FUNCTION_BLOCK EM_LogicExample_1 EXTENDS FB_EM_Base IMPLEMENTS ITF_EM_LogicExample1
VAR_INPUT	
	i_stMachineCommands				: ST_UN_Machine100_Cmd;
END_VAR
VAR
// Variables
	s_bStaStateOfSomething			: BOOL;
	s_bStaStateOfSomething2			: BOOL;
	s_bStaStateOfSomething3			: BOOL;
	s_bStaStateOfSomething4			: BOOL;
	s_bStaStateOfSomething5			: BOOL;
	s_bStaStateOfSomething6			: BOOL;
	s_bStaStateOfSomething7			: BOOL;
	s_fStaValue						: LREAL;
	s_fStaValueResult				: LREAL;
	
// Config Struct
	s_stConfig						: ST_EM_LogicExample1_Config;
	
// Control modules
	s_cmVirtualMaster				: CM_Servo_Virtual;
	s_cmAxis1						: CM_Servo_Virtual;
	s_cmAxis1Cam					: CM_Servo_CammingAddon(s_cmAxis1);
	s_cmAxis1Fly					: CM_Servo_FlyingSawAddon(s_cmAxis1);
	s_cmWaterInlet					: CM_Valve;
	s_cmBelt						: CM_MotorDol;
	s_cmHeightAdjuster				: CM_MotorDol_AF;
	s_cmVentilator					: CM_MotorVFD_Lenze_i5xx;
	
// Inputs
	s_fbDiSensorPos1				: FB_DigitalInput;
	
// Outputs
	s_fbDoMachineX_Start			: FB_DigitalOutput;
	s_fbAoMachineX_Speed			: FB_AnalogOutput;
	s_fbRedLight					: FB_Light;
	s_fbBlueButton					: FB_PushButtonLight;
	s_fbStackLight					: FB_StackLights;
	
// Alarms
	s_AlmFailure1					: FB_AlarmHandler;
	s_AlmFailure2					: FB_AlarmHandler;
	
// Statistics
	s_fbRunTime_Belt				: FB_RunningTime;
	
END_VAR
VAR CONSTANT
	nCamTableIdAxis1			: UINT := 1;
END_VAR

SUPER^();

METHOD PROTECTED _m_Aborting
VAR_INPUT
	i_rstPML_Status			: REFERENCE TO ST_PackML_Status;
END_VAR
VAR_INST
	
	s_bStaStateComplete1		: BOOL;
END_VAR
i_rstPML_Status.bStateComplete := _m_StopServos(i_bReqStart := i_rstPML_Status.bStateEntry);
END_METHOD

METHOD PROTECTED _m_Alarms
VAR_INST
	s_tonAlmFailure2_DelayedAutoReset	: TON;
END_VAR
SUPER^._m_Alarms();

// Failure 1
s_stConfig.stAlmFailure1.nIDnr		:= 1;
s_stConfig.stAlmFailure1.eAction	:= E_Alarm_Actions.Abort;
s_stConfig.stAlmFailure1.tmDelay	:= T#1S;
s_stConfig.stAlmFailure1.bEnable	:= q_bStaEnabled;
s_AlmFailure1(
	i_bCmdSet	:= s_fbDiSensorPos1.q_bStaInput 
				AND s_bStaStateOfSomething,
	i_sMsgVar1	:= 'Fault code: ',
	//i_sMsgVar2	:= TO_STRING(s_nFaultCode),
	i_rstConfig	:= s_stConfig.stAlmFailure1,
	i_itfAlarmCollector := s_fbAlarmCollector);

	
// Failure 2
s_stConfig.stAlmFailure2.nIDnr	:= 2;
s_stConfig.stAlmFailure2.eAction := E_Alarm_Actions.Suspend;

// Automatic reset timer
s_tonAlmFailure2_DelayedAutoReset(IN := s_AlmFailure2.p_bStaActive AND NOT s_AlmFailure2.p_bStaCmdSet, PT := T#5S);
// Reset the alarm after the delay time
IF s_tonAlmFailure2_DelayedAutoReset.Q THEN
	s_AlmFailure2.m_CmdReset();
END_IF

s_AlmFailure2(
	i_rstConfig	:= s_stConfig.stAlmFailure2,
	i_itfAlarmCollector := s_fbAlarmCollector);
END_METHOD

METHOD PROTECTED _m_Execute
VAR_INPUT
	i_rstPML_Status			: REFERENCE TO ST_PackML_Status;
END_VAR
VAR_INST
	s_eActMode				: E_PackML_Mode;
END_VAR
// Execute only when in a specific mode
s_eActMode := i_rstPML_Status.eActMode;
CASE s_eActMode OF
	E_PackML_Mode.Production: 
		// Execute only when in PRODUCTION mode
		i_rstPML_Status.bStateComplete := _m_Execute_Production(i_bReqStart := i_rstPML_Status.bStateEntry);
				
ELSE
	// Execute in all other modes	
	i_rstPML_Status.bStateComplete := TRUE;
END_CASE
END_METHOD

METHOD PROTECTED _m_Execute_Production : BOOL
VAR_INPUT
	i_bReqStart				: BOOL;
END_VAR
VAR_INST
	s_fbSeqControl			: FB_SeqControl;
	s_eSeqAutoExecute		: E_EM_LogicExample1_Seq_ExecuteProduction;
	s_stSyncMode			: ST_SyncMode;			// Synchronisation mode
	
	
	s_fCalculatedSpeed		: LREAL;		// Calculated VM speed, based on machine setting
	s_fShortestPosition		: LREAL;		
END_VAR
// Sequence exceptions
// n.a.


// Sequencer control
s_fbSeqControl(
	i_bReqStart		:= i_bReqStart, 
	i_rnActSeqStep	:= s_eSeqAutoExecute,
	i_sActSeqStep	:= TO_STRING(s_eSeqAutoExecute));
	
// Sequence	
CASE s_eSeqAutoExecute OF
	
	E_EM_LogicExample1_Seq_ExecuteProduction.Idle:
		;
			
	E_EM_LogicExample1_Seq_ExecuteProduction.Start:
		s_fCalculatedSpeed	:= (360.0 * 1000.0) / 123.4; // 360 degree = 1 product. 
		IF s_cmVirtualMaster.m_StartFF(
			i_bCmdReset		:= s_fbSeqControl.q_bStaEntry, 
			i_fAcceleration	:= s_cmVirtualMaster.q_stParameterSet.fAccelerationMax, 
			i_fDeceleration	:= s_cmVirtualMaster.q_stParameterSet.fDecelerationMax, 
			i_fJerk			:= s_cmVirtualMaster.q_stParameterSet.fJerk, 
			i_fSpeed		:= s_cmVirtualMaster.q_stParameterSet.fVeloFastManual,
			i_sLogHint		:= '',
			i_eBufferMode	:= MC_BufferMode.MC_Aborting) 
		THEN
			s_fbSeqControl.m_ReqStep(E_EM_LogicExample1_Seq_ExecuteProduction.StartWait);
		END_IF
		

	//Wait for 5 seconds
	E_EM_LogicExample1_Seq_ExecuteProduction.StartWait:
		IF s_fbSeqControl.q_tmStepTime> T#5S THEN
			s_fbSeqControl.m_ReqStep(E_EM_LogicExample1_Seq_ExecuteProduction.Step1);
		END_IF

		
	//gear out Slave axis 1 without stopping the axis
	E_EM_LogicExample1_Seq_ExecuteProduction.Step1:
		IF s_cmAxis1.m_GearOut(i_bCmdReset:=s_fbSeqControl.q_bStaEntry) THEN
			s_fbSeqControl.m_ReqStep(E_EM_LogicExample1_Seq_ExecuteProduction.Step1Wait);
		END_IF

		
	//Wait for 5 seconds
	E_EM_LogicExample1_Seq_ExecuteProduction.Step1Wait:
		IF s_fbSeqControl.q_tmStepTime> T#5S THEN
			s_fbSeqControl.m_ReqStep(E_EM_LogicExample1_Seq_ExecuteProduction.Step2);
		END_IF
		
		
	//gear in Slave axis 1 at position
	E_EM_LogicExample1_Seq_ExecuteProduction.Step2:
		IF s_fbSeqControl.q_bStaEntry THEN
			//Enable disable checks. An enabled check gives an NC error when the check condition is true.	
			s_stSyncMode.GearInSyncMode 						:= E_GearInSyncMode.GEARINSYNCMODE_POSITIONBASED;
			s_stSyncMode.GearInSync_CheckMask_MinPos 			:= FALSE;
			s_stSyncMode.GearInSync_CheckMask_MaxPos 			:= FALSE;
			s_stSyncMode.GearInSync_CheckMask_MaxVelo 			:= FALSE;
			s_stSyncMode.GearInSync_CheckMask_MaxAcc 			:= FALSE;
			s_stSyncMode.GearInSync_CheckMask_MaxDec 			:= FALSE;
			s_stSyncMode.GearInSync_CheckMask_MaxJerk 			:= FALSE;
			s_stSyncMode.GearInSync_CheckMask_OvershootPos 		:= FALSE;
			s_stSyncMode.GearInSync_CheckMask_UndershootPos 	:= FALSE;
			s_stSyncMode.GearInSync_CheckMask_OvershootVelo 	:= FALSE;
			s_stSyncMode.GearInSync_CheckMask_UndershootVelo 	:= FALSE;
			s_stSyncMode.GearInSync_CheckMask_OvershootVeloZero := FALSE;
			s_stSyncMode.GearInSync_CheckMask_UndershootVeloZero:= FALSE;
			
			//Optimalization methodes
			s_stSyncMode.GearInSync_OpMask_RollbackLock 		:= TRUE;
			s_stSyncMode.GearInSync_OpMask_InstantStopOnRollback:= TRUE;
			s_stSyncMode.GearInSync_OpMask_PreferConstVelo 		:= TRUE;
			s_stSyncMode.GearInSync_OpMask_IgnoreMasterAcc 		:= TRUE;
		END_IF

		IF s_cmAxis1Fly.m_GearInPos(
			i_bCmdReset				:= s_fbSeqControl.q_bStaEntry, 
			i_fAcceleration			:= s_cmAxis1.q_stParameterSet.fAccelerationMax, 
			i_fDeceleration			:= s_cmAxis1.q_stParameterSet.fDecelerationMax, 
			i_fJerk					:= s_cmAxis1.q_stParameterSet.fJerk, 
			i_fSpeed				:= s_cmAxis1.q_stParameterSet.fVeloMaximum, 
			i_fMasterSyncPosition	:= s_cmVirtualMaster.q_fActualPos + 1000.0, 
			i_fSlaveSyncPosition	:= s_cmAxis1.q_fActualPos + 2000.0, 
			i_stSyncMode			:= s_stSyncMode, 
			i_fSlaveScale			:= 1.0, 
			i_fMasterScale			:= 1.0, 
			i_itfMaster				:= s_cmVirtualMaster) 
		THEN
			s_fbSeqControl.m_ReqStep(E_EM_LogicExample1_Seq_ExecuteProduction.Step2Wait);
		END_IF

		
	//Wait till synchronized
	E_EM_LogicExample1_Seq_ExecuteProduction.Step2Wait:
		IF s_cmAxis1.q_bStaInSync THEN
			s_fbSeqControl.m_ReqStep(E_EM_LogicExample1_Seq_ExecuteProduction.Step3);
		END_IF
		
		
	//gear out Slave axis 1 without stopping the axis when the axis is synchronized
	E_EM_LogicExample1_Seq_ExecuteProduction.Step3:
		IF s_cmAxis1.m_GearOut(i_bCmdReset:=s_fbSeqControl.q_bStaEntry) THEN
			s_fbSeqControl.m_ReqStep(E_EM_LogicExample1_Seq_ExecuteProduction.Step3Wait);
		END_IF

		
	//Wait for 5 seconds
	E_EM_LogicExample1_Seq_ExecuteProduction.Step3Wait:
		IF s_fbSeqControl.q_tmStepTime> T#5S THEN
			s_fbSeqControl.m_ReqStep(E_EM_LogicExample1_Seq_ExecuteProduction.Step4);
		END_IF
		
		
	//gear in Slave axis 1 at speed
	E_EM_LogicExample1_Seq_ExecuteProduction.Step4:
		IF s_fbSeqControl.q_bStaEntry THEN
			//Enable disable checks. An enabled check gives an NC error when the check condition is true.	
			s_stSyncMode.GearInSyncMode 						:= E_GearInSyncMode.GEARINSYNCMODE_POSITIONBASED;
			s_stSyncMode.GearInSync_CheckMask_MinPos 			:= FALSE;
			s_stSyncMode.GearInSync_CheckMask_MaxPos 			:= FALSE;
			s_stSyncMode.GearInSync_CheckMask_MaxVelo 			:= FALSE;
			s_stSyncMode.GearInSync_CheckMask_MaxAcc 			:= FALSE;
			s_stSyncMode.GearInSync_CheckMask_MaxDec 			:= FALSE;
			s_stSyncMode.GearInSync_CheckMask_MaxJerk 			:= FALSE;
			s_stSyncMode.GearInSync_CheckMask_OvershootPos 		:= FALSE;
			s_stSyncMode.GearInSync_CheckMask_UndershootPos 	:= FALSE;
			s_stSyncMode.GearInSync_CheckMask_OvershootVelo 	:= FALSE;
			s_stSyncMode.GearInSync_CheckMask_UndershootVelo 	:= FALSE;
			s_stSyncMode.GearInSync_CheckMask_OvershootVeloZero := FALSE;
			s_stSyncMode.GearInSync_CheckMask_UndershootVeloZero:= FALSE;
			
			//Optimalization methodes
			s_stSyncMode.GearInSync_OpMask_RollbackLock 		:= TRUE;
			s_stSyncMode.GearInSync_OpMask_InstantStopOnRollback:= TRUE;
			s_stSyncMode.GearInSync_OpMask_PreferConstVelo 		:= TRUE;
			s_stSyncMode.GearInSync_OpMask_IgnoreMasterAcc 		:= TRUE;
		END_IF
	
		IF s_cmAxis1Fly.m_GearInSpeed(
			i_bCmdReset		:= s_fbSeqControl.q_bStaEntry, 
			i_fSlaveScale	:= 2.0, 
			i_fMasterScale	:= 1.0, 
			i_stSyncMode	:= s_stSyncMode, 
			i_fAcceleration	:= s_cmAxis1.q_stParameterSet.fAccelerationMax, 
			i_fDeceleration	:= s_cmAxis1.q_stParameterSet.fDecelerationMax, 
			i_fJerk			:= s_cmAxis1.q_stParameterSet.fJerk, 
			i_fSpeed		:= s_cmAxis1.q_stParameterSet.fVeloMaximum, 
			i_itfMaster		:= s_cmVirtualMaster ) 
		THEN
			s_fbSeqControl.m_ReqStep(E_EM_LogicExample1_Seq_ExecuteProduction.Step4Wait);
		END_IF

		
	//Wait till synchronized
	E_EM_LogicExample1_Seq_ExecuteProduction.Step4Wait:
		IF s_cmAxis1.q_bStaInSync THEN
			s_fbSeqControl.m_ReqStep(E_EM_LogicExample1_Seq_ExecuteProduction.Step5);
		END_IF
		
		
	//halt Master and Slave axis => axis will gearout and stopping 
	E_EM_LogicExample1_Seq_ExecuteProduction.Step5:
			IF s_cmVirtualMaster.m_Halt(
				i_bCmdReset		:= s_fbSeqControl.q_bStaEntry,
				i_fDeceleration	:= s_cmVirtualMaster.q_stParameterSet.fDecelerationMax,
				i_fJerk			:= s_cmVirtualMaster.q_stParameterSet.fJerk,
				i_eBufferMode	:= MC_BufferMode.MC_Aborting) 
			AND
				s_cmAxis1.m_Halt(
				i_bCmdReset		:= s_fbSeqControl.q_bStaEntry,
				i_fDeceleration	:= s_cmAxis1.q_stParameterSet.fDecelerationMax,
				i_fJerk			:= s_cmAxis1.q_stParameterSet.fJerk, 
				i_eBufferMode	:= MC_BufferMode.MC_Aborting) 
			THEN
			s_fbSeqControl.m_ReqStep(E_EM_LogicExample1_Seq_ExecuteProduction.Step5Wait);
			END_IF

			
	//Wait till axis standstill
	E_EM_LogicExample1_Seq_ExecuteProduction.Step5Wait:
		IF s_cmAxis1.q_stAxisState.StandStill AND s_cmVirtualMaster.q_stAxisState.StandStill THEN
			s_fbSeqControl.m_ReqStep(E_EM_LogicExample1_Seq_ExecuteProduction.Step6);
		END_IF
			
		
	//Gear in dynamic 
	E_EM_LogicExample1_Seq_ExecuteProduction.Step6:
		IF s_cmAxis1.m_GearInDyn(
			i_bCmdReset		:= s_fbSeqControl.q_bStaEntry, 
			i_fAcceleration	:= s_cmAxis1.q_stParameterSet.fAccelerationMax, 
			i_fDeceleration	:= s_cmAxis1.q_stParameterSet.fDecelerationMax, 
			i_fJerk			:= s_cmAxis1.q_stParameterSet.fJerk, 
			i_fGearRatio	:= 1.0, 
			i_itfMaster		:= s_cmVirtualMaster) 
		THEN
			//No wait step nessary m_GearInDyn give TRUE when axis is coupled
			s_fbSeqControl.m_ReqStep(E_EM_LogicExample1_Seq_ExecuteProduction.Step7);
		END_IF
		
	//Move master relative 
	E_EM_LogicExample1_Seq_ExecuteProduction.Step7:
		IF s_cmVirtualMaster.m_StartRelative(
			i_bCmdReset		:= s_fbSeqControl.q_bStaEntry, 
			i_fAcceleration	:= s_cmVirtualMaster.q_stParameterSet.fAccelerationMax, 
			i_fDeceleration	:= s_cmVirtualMaster.q_stParameterSet.fDecelerationMax, 
			i_fJerk			:= s_cmVirtualMaster.q_stParameterSet.fJerk, 
			i_fSpeed		:= s_cmVirtualMaster.q_stParameterSet.fVeloFastManual, 
			i_fPosition		:= 1000.0,
			i_sLogHint		:= '',
			i_eBufferMode	:= MC_BufferMode.MC_Aborting) 
		THEN
			s_fbSeqControl.m_ReqStep(E_EM_LogicExample1_Seq_ExecuteProduction.Step7Wait);
		END_IF

		
	//Wait for 5 seconds
	E_EM_LogicExample1_Seq_ExecuteProduction.Step7Wait:
		IF s_fbSeqControl.q_tmStepTime> T#5S THEN
			s_fbSeqControl.m_ReqStep(E_EM_LogicExample1_Seq_ExecuteProduction.Step8);
		END_IF
		
		
	//Change gearfactor 
	E_EM_LogicExample1_Seq_ExecuteProduction.Step8:
		IF s_cmAxis1.m_GearInDynGearRatio(i_fGearRatio:= 0.5) THEN
			s_fbSeqControl.m_ReqStep(E_EM_LogicExample1_Seq_ExecuteProduction.Step8Wait);
		END_IF

		
	//Wait for 5 seconds
	E_EM_LogicExample1_Seq_ExecuteProduction.Step8Wait:
		IF s_fbSeqControl.q_tmStepTime> T#5S THEN
			s_fbSeqControl.m_ReqStep(E_EM_LogicExample1_Seq_ExecuteProduction.Step9);
		END_IF
		
		
	//stop Master and Slave axis => axis will gearout and stopping 
	E_EM_LogicExample1_Seq_ExecuteProduction.Step9:
		IF s_cmVirtualMaster.m_Stop(
			i_bCmdReset		:= s_fbSeqControl.q_bStaEntry,
			i_fDeceleration	:= s_cmVirtualMaster.q_stParameterSet.fDecelerationMax,
			i_fJerk			:= s_cmVirtualMaster.q_stParameterSet.fJerk) 
		AND
			s_cmAxis1.m_Stop(
			i_bCmdReset		:= s_fbSeqControl.q_bStaEntry,
			i_fDeceleration	:= s_cmAxis1.q_stParameterSet.fDecelerationMax,
			i_fJerk			:= s_cmAxis1.q_stParameterSet.fJerk) 
		THEN
			s_fbSeqControl.m_ReqStep(E_EM_LogicExample1_Seq_ExecuteProduction.Step10Wait);
		END_IF

		
	//Wait till axis standstill
	E_EM_LogicExample1_Seq_ExecuteProduction.Step10Wait:
		IF s_cmAxis1.q_stAxisState.StandStill AND s_cmVirtualMaster.q_stAxisState.StandStill THEN
			s_fbSeqControl.m_ReqStep(E_EM_LogicExample1_Seq_ExecuteProduction.Step11);
		END_IF
		
		
	//Gear in static 
	E_EM_LogicExample1_Seq_ExecuteProduction.Step11:
		IF s_cmAxis1.m_GearInStatic(
			i_bCmdReset		:= s_fbSeqControl.q_bStaEntry, 
			i_fAcceleration	:= s_cmAxis1.q_stParameterSet.fAccelerationMax, 
			i_fDeceleration	:= s_cmAxis1.q_stParameterSet.fDecelerationMax, 
			i_fJerk			:= s_cmAxis1.q_stParameterSet.fJerk, 
			i_fSlaveScale	:= 1.0,
			i_fMasterScale	:= 1.0, 
			i_itfMaster		:= s_cmVirtualMaster) 
		THEN
			//No wait step nessary m_GearInStatic give TRUE when axis is coupled
			s_fbSeqControl.m_ReqStep(E_EM_LogicExample1_Seq_ExecuteProduction.Step12);
		END_IF
		
		
	//Move master reverse 
	E_EM_LogicExample1_Seq_ExecuteProduction.Step12:
		IF s_cmVirtualMaster.m_StartRev(
			i_bCmdReset		:= s_fbSeqControl.q_bStaEntry, 
			i_fAcceleration	:= s_cmVirtualMaster.q_stParameterSet.fAccelerationMax, 
			i_fDeceleration	:= s_cmVirtualMaster.q_stParameterSet.fDecelerationMax, 
			i_fJerk			:= s_cmVirtualMaster.q_stParameterSet.fJerk, 
			i_fSpeed		:= s_cmVirtualMaster.q_stParameterSet.fVeloFastManual,
			i_sLogHint		:= '',
			i_eBufferMode	:= MC_BufferMode.MC_Aborting) 
		THEN
			s_fbSeqControl.m_ReqStep(E_EM_LogicExample1_Seq_ExecuteProduction.Step12Wait);
		END_IF

		
	//Wait for 5 seconds
	E_EM_LogicExample1_Seq_ExecuteProduction.Step12Wait:
		IF s_fbSeqControl.q_tmStepTime> T#5S THEN
			s_fbSeqControl.m_ReqStep(E_EM_LogicExample1_Seq_ExecuteProduction.Step13);
		END_IF
		
		
	//stop only the slave axis and move the master axis forward
	E_EM_LogicExample1_Seq_ExecuteProduction.Step13:
		IF s_cmAxis1.m_Halt(
			i_bCmdReset		:= s_fbSeqControl.q_bStaEntry,
			i_fDeceleration	:= s_cmAxis1.q_stParameterSet.fDecelerationMax,
			i_fJerk			:= s_cmAxis1.q_stParameterSet.fJerk,
			i_eBufferMode	:= MC_BufferMode.MC_Aborting) 
		AND s_cmVirtualMaster.m_StartFF(
			i_bCmdReset		:= s_fbSeqControl.q_bStaEntry, 
			i_fAcceleration	:= s_cmVirtualMaster.q_stParameterSet.fAccelerationMax, 
			i_fDeceleration	:= s_cmVirtualMaster.q_stParameterSet.fDecelerationMax, 
			i_fJerk			:= s_cmVirtualMaster.q_stParameterSet.fJerk, 
			i_fSpeed		:= s_cmVirtualMaster.q_stParameterSet.fVeloFastManual,
			i_sLogHint		:= '',
			i_eBufferMode	:= MC_BufferMode.MC_Aborting) 
		THEN
			s_fbSeqControl.m_ReqStep(E_EM_LogicExample1_Seq_ExecuteProduction.Step13Wait);
		END_IF

		
	//Wait for 5 seconds
	E_EM_LogicExample1_Seq_ExecuteProduction.Step13Wait:
		IF s_fbSeqControl.q_tmStepTime> T#5S THEN
			s_fbSeqControl.m_ReqStep(E_EM_LogicExample1_Seq_ExecuteProduction.Step14);
		END_IF
		
		
	//stop master axis
	E_EM_LogicExample1_Seq_ExecuteProduction.Step14:
		IF s_cmVirtualMaster.m_Halt(
			i_bCmdReset		:= s_fbSeqControl.q_bStaEntry,
			i_fDeceleration	:= s_cmVirtualMaster.q_stParameterSet.fDecelerationMax,
			i_fJerk			:= s_cmVirtualMaster.q_stParameterSet.fJerk,
			i_eBufferMode	:= MC_BufferMode.MC_Aborting) 
		THEN
			s_fbSeqControl.m_ReqStep(E_EM_LogicExample1_Seq_ExecuteProduction.Step14Wait);
		END_IF

		
	//Wait till axis standstill
	E_EM_LogicExample1_Seq_ExecuteProduction.Step14Wait:
		IF s_cmVirtualMaster.q_stAxisState.StandStill THEN
			s_fbSeqControl.m_ReqStep(E_EM_LogicExample1_Seq_ExecuteProduction.Step15);
		END_IF
		
		
	//set both axis to zero
	E_EM_LogicExample1_Seq_ExecuteProduction.Step15:
		IF s_cmVirtualMaster.m_SetActualPosition(
			i_bCmdReset := s_fbSeqControl.q_bStaEntry,
			i_fPosition	:= 0)
		AND
			s_cmAxis1.m_SetActualPosition(
			i_bCmdReset := s_fbSeqControl.q_bStaEntry,
			i_fPosition	:= 0)
		THEN
			// No Cam-license available
			//s_fbSeqControl.m_ReqStep(E_EM_LogicExample1_Seq_AutoExecute.Step16);
			s_fbSeqControl.m_ReqStep(E_EM_LogicExample1_Seq_ExecuteProduction.Step17);
		END_IF

		
	//Cam in slave to master 
	E_EM_LogicExample1_Seq_ExecuteProduction.Step16:
		IF s_cmAxis1Cam.m_CamIn(
				i_bCmdReset					:= s_fbSeqControl.q_bStaEntry,
				i_fMasterOffset				:= 0.0,
				i_fSlaveOffset				:= 0.0,
				i_fMasterScale				:= 1,
				i_fSlaveScale				:= 1,
				i_bMasterOffsetIsRelative	:= FALSE,
				i_bSlaveOffsetIsRelative	:= FALSE,
				i_nCamTableId				:= nCamTableIdAxis1, 
				i_fMasterActivationPos		:= 0, 
				i_mcCamOperationMode		:= MC_CamOperationMode.CAMOPERATIONMODE_EXCHANGE,
				i_nReferenceCamTableID		:= 0,
				i_mcCamActivationMode		:= MC_CamActivationMode.MC_CAMACTIVATION_INSTANTANEOUS,
				i_mcMasterScalingMode		:= MC_CamScalingMode.MC_CAMSCALING_USERDEFINED,
				i_mcSlaveScalingMode		:= MC_CamScalingMode.MC_CAMSCALING_USERDEFINED,
				i_itfMaster					:= s_cmVirtualMaster)
		THEN
			s_fbSeqControl.m_ReqStep(E_EM_LogicExample1_Seq_ExecuteProduction.Step17);
		END_IF

		
	//Move absolute
	E_EM_LogicExample1_Seq_ExecuteProduction.Step17:
		s_fCalculatedSpeed	:= (360.0 * 100.0) / 123.4; // 360 degree = 1 product. 
		IF s_cmVirtualMaster.m_StartAbsolute(
				i_bCmdReset		:= s_fbSeqControl.q_bStaEntry,
				i_fAcceleration	:= s_cmVirtualMaster.q_stParameterSet.fAcceleration,
				i_fDeceleration	:= s_cmVirtualMaster.q_stParameterSet.fDeceleration,
				i_fJerk			:= s_cmVirtualMaster.q_stParameterSet.fJerk,
				i_fSpeed		:= s_fCalculatedSpeed,
				i_fPosition		:= TO_LREAL(s_cmVirtualMaster.q_nCommandedTurnsModulo+1) * 360.0, //Move 1 modulo position forwards 
				i_eBufferMode	:= MC_BufferMode.MC_Aborting, 
				i_sLogHint		:= 'Takt' )
		THEN
			s_fbSeqControl.m_ReqStep(E_EM_LogicExample1_Seq_ExecuteProduction.Start);
		END_IF
		
		
	//Stop both axis when execute is finished	
	E_EM_LogicExample1_Seq_ExecuteProduction.StopAxis:
		IF s_cmVirtualMaster.m_Stop(
			i_bCmdReset		:= s_fbSeqControl.q_bStaEntry,
			i_fDeceleration	:= s_cmVirtualMaster.q_stParameterSet.fDecelerationMax,
			i_fJerk			:= s_cmVirtualMaster.q_stParameterSet.fJerk) 
		AND
			s_cmAxis1.m_Stop(
			i_bCmdReset		:= s_fbSeqControl.q_bStaEntry,
			i_fDeceleration	:= s_cmAxis1.q_stParameterSet.fDecelerationMax,
			i_fJerk			:= s_cmAxis1.q_stParameterSet.fJerk) 
		THEN
			s_fbSeqControl.m_ReqStep(E_EM_LogicExample1_Seq_ExecuteProduction.WaitStopAxis);
		END_IF

		
	//Wait till both axis are stopped
	E_EM_LogicExample1_Seq_ExecuteProduction.WaitStopAxis:	
		IF s_cmVirtualMaster.q_stAxisState.StandStill AND s_cmAxis1.q_stAxisState.StandStill THEN
			s_fbSeqControl.m_ReqStep(E_EM_LogicExample1_Seq_ExecuteProduction.Ready);
		END_IF	
		
		
	E_EM_LogicExample1_Seq_ExecuteProduction.Ready:
		;
		
		
	E_EM_LogicExample1_Seq_ExecuteProduction.Error:
		;
END_CASE

// Sequence state to PackML commands
F_SeqControl_PackMLcommands(
	i_rnActSeqStep	:= s_eSeqAutoExecute,
	q_bStaFinished	=> _m_Execute_Production,
	q_bStaIdle		=> ,
	q_bStaError		=> );
END_METHOD

METHOD PROTECTED _m_Init
SUPER^._m_Init();

// Do some initializations here..


// Failure 1
s_stConfig.stAlmFailure1.eAction := E_Alarm_Actions.Abort;
s_stConfig.stAlmFailure1.tmDelay := T#1S;
END_METHOD

METHOD PROTECTED _m_Inputs
SUPER^._m_Inputs();

// Simulation
IF s_fbSimulation.q_bStaOn THEN
	s_fbDiSensorPos1.m_SimulationOn(i_bValue := TRUE);
ELSIF s_fbSimulation.q_bStaOsf THEN
	s_fbDiSensorPos1.m_SimulationOff();
END_IF

// Sensor at position 1
s_stConfig.stDiSensorPos1.bCfgInvert	:= TRUE;
s_stConfig.stDiSensorPos1.tmOnDelay		:= T#50MS;
s_fbDiSensorPos1(i_rstConfig := s_stConfig.stDiSensorPos1);

// Blue button with light
s_fbBlueButton(
	i_bReqLightOn		:= s_fbBlueButton.q_bStaInput, 
	i_bReqFlashLight	:= s_bStaStateOfSomething, 
	i_rstConfig			:= s_stConfig.stBlueButton);
END_METHOD

METHOD PROTECTED _m_Logic
VAR_INST
	s_osrStateOfSomething	: R_TRIG;
END_VAR
SUPER^._m_Logic();

// ============ Enable parts of the EM ============
// Allow manual control from HMI when the actual mode is 'Manual' and actual state is 'Execute'
s_bAlwManualControl	:= s_stPML.stStatus.eActMode = E_PackML_Mode.Manual 
					AND s_stPML.stStatus.eActState = E_PackML_State.Execute;

// Allow alarming when module is enabled
s_bReqAlarmCollector_Enable := s_bStaEnable;

// Allow PackML when module is enabled. 
s_stPML.stConfig.bEnabled := s_bStaEnable;

// ============ Statusses ============
// Status updated in every mode and every state
s_bStaStateOfSomething := s_cmWaterInlet.q_bStaOff AND s_cmAxis1.q_bStaInPos;
s_osrStateOfSomething(CLK := s_bStaStateOfSomething);


// Set alarm when s_bStaStateOfSomething3 is active
IF s_bStaStateOfSomething3 AND GVL_GBL.g_fbSystem.p_bPulse1Hz THEN
	s_AlmFailure2.m_CmdSet('Text1','Text2','Text3');
END_IF

// ============ Logging ============
// Log state continuously, Fills the log quickly...
IF s_osrStateOfSomething.Q THEN
	(* Logging *)
	g_fbGBL_Logger.m_InitLogString(
		i_sInstance := s_sInstance, 
		i_sMethode := 'm_Logic', 
		i_sFunction := '', 
		i_sDescription := '');	
	g_fbGBL_Logger.m_AddBoolParam('s_bStaStateOfSomething',s_bStaStateOfSomething2);
	g_fbGBL_Logger.m_WriteLogString(i_eSeverity := E_LogSeverity.Fatal);
END_IF


s_fStaValueResult := F_fCalcFloorModuloPosition(i_fActualPosition := s_fStaValue, i_fMod := 360.0);

IF s_bStaStateOfSomething4 THEN
	F_ProgramError_Set(
		i_sInstancePath	:= s_sInstance,
		i_sMsgVar1	:= 'text1',
		i_sMsgVar2	:= 'text2',
		i_sMsgVar3	:= 'text3');
END_IF
END_METHOD

METHOD PROTECTED _m_Modules
SUPER^._m_Modules();

// Virtual Master
s_cmVirtualMaster(
	i_bReqEnable				:= s_bStaEnable, 
	i_bReqReset					:= s_fbAlarmCollector.q_bReqReset,
	i_bAlwManualCtrl			:= s_bAlwManualControl,
	i_bReqSimulationOn			:= s_fbSimulation.q_bStaOn,
	i_sPostFixAlarmValueMessage	:= 'Virtual master',
	i_itfAlarmCollector_Parent	:= s_fbAlarmCollector, 
	i_rstConfig					:= s_stConfig.stCmVirtualMaster, 
	i_bEmrStopOk				:= i_bStaSafetyOk, 
	i_fOverride					:= 100.0, 
	i_bDisableForward			:= FALSE, 
	i_bDisableReverse			:= FALSE, 
	i_bDisableAxis				:= FALSE);


// Servo axis 1
s_stConfig.stCmAxis1.tmReferenceTimeOut	:= T#1M;
s_cmAxis1(
	i_bReqEnable				:= s_bStaEnable, 
	i_bReqReset					:= s_fbAlarmCollector.q_bReqReset,
	i_bAlwManualCtrl			:= s_bAlwManualControl,
	i_bReqSimulationOn			:= s_fbSimulation.q_bStaOn,
	i_sPostFixAlarmValueMessage	:= 'Mover axis 1',
	i_itfAlarmCollector_Parent	:= s_fbAlarmCollector,  
	i_rstConfig					:= s_stConfig.stCmAxis1, 
	i_bEmrStopOk				:= i_bStaSafetyOk, 
	i_fOverride					:= 100.0, 
	i_bDisableForward			:= FALSE, 
	i_bDisableReverse			:= FALSE, 
	i_bDisableAxis				:= FALSE);

// Valve 1
s_stConfig.stCmValve1.stAlarmCollector.eSubstituteActionForPackML_Abort := E_Alarm_Actions.NoAction;
s_stConfig.stCmValve1.stHardware.nCfgFeedbackOn := 0;
s_stConfig.stCmValve1.stHardware.nCfgFeedbackOff := 0;
s_stConfig.stCmValve1.stAlmBothOn.tmDelay	:= T#100MS;
s_cmWaterInlet(
	i_bReqEnable		:= s_bStaEnable, 
	i_bReqReset			:= s_fbAlarmCollector.q_bReqReset,
	i_bAlwManualCtrl	:= s_bAlwManualControl,
	i_bReqSimulationOn	:= s_fbSimulation.q_bStaOn,
	i_itfAlarmCollector_Parent	:= s_fbAlarmCollector,  
	i_rstConfig			:= s_stConfig.stCmValve1);

// Motor DOL 1
s_cmBelt(
	i_bReqEnable		:= s_bStaEnable, 
	i_bReqReset			:= s_fbAlarmCollector.q_bReqReset, 
	i_bAlwManualCtrl	:= s_bAlwManualControl,
	i_bReqSimulationOn	:= s_fbSimulation.q_bStaOn,
	i_itfAlarmCollector_Parent	:= s_fbAlarmCollector,  
	i_rstConfig			:= s_stConfig.stCmMotorDol1);
	
// Motor DOL with analog position feedback 1
s_cmHeightAdjuster(
	i_bReqEnable		:= s_bStaEnable, 
	i_bReqReset			:= s_fbAlarmCollector.q_bReqReset, 
	i_bAlwManualCtrl	:= s_bAlwManualControl, 
	i_bReqSimulationOn	:= s_fbSimulation.q_bStaOn,
	i_itfAlarmCollector_Parent	:= s_fbAlarmCollector,  
	i_rstConfig			:= s_stConfig.stCmMotorDolAF1.stCmMotorDol,
	i_rstConfig_AF		:= s_stConfig.stCmMotorDolAF1);	
	

// Ventilator motor with Lenze i550 drive
s_stConfig.stCmVentilator.bAllowReverse := TRUE;
// Motor params to drive
s_stConfig.stCmVentilator.astMotorParameter[0].fLocalPar := 0.81;		// [kW] Rated Power		
s_stConfig.stCmVentilator.astMotorParameter[1].fLocalPar := 1375.0;     // [rpm] Rated Speed		
s_stConfig.stCmVentilator.astMotorParameter[2].fLocalPar := 0.51;       // [A] Rated Current		
s_stConfig.stCmVentilator.astMotorParameter[3].fLocalPar := 400.0;      // [V] Rated Voltage		
s_stConfig.stCmVentilator.astMotorParameter[4].fLocalPar := 50.0;       // [Hz] Rated Frequency	
s_stConfig.stCmVentilator.astMotorParameter[5].fLocalPar := 0.65;       // [] Cosine Phi			
s_stConfig.stCmVentilator.astMotorParameter[6].fLocalPar := 3000.0;     // [rpm] Max Speed			
// Drive params to drive
s_stConfig.stCmVentilator.astDriveParameters[4].nData := 49; // Configure Control word bit 1 as "Release Holding Brake"
s_cmVentilator(
	i_bReqEnable		:= s_bStaEnable, 
	i_bReqReset			:= s_fbAlarmCollector.q_bReqReset, 
	i_bAlwManualCtrl	:= s_bAlwManualControl, 
	i_bReqSimulationOn	:= s_fbSimulation.q_bStaOn,
	i_itfAlarmCollector_Parent	:= s_fbAlarmCollector,  
	i_rstConfig			:= s_stConfig.stCmVentilator);
END_METHOD

METHOD PROTECTED _m_Outputs
SUPER^._m_Outputs();

// Simulation
IF s_fbSimulation.q_bStaOsr THEN
	s_fbDoMachineX_Start.m_SimulationOn();
	s_fbAoMachineX_Speed.m_SimulationOn();
ELSIF s_fbSimulation.q_bStaOsf THEN
	s_fbDoMachineX_Start.m_SimulationOff();
	s_fbAoMachineX_Speed.m_SimulationOff();
END_IF

// Machine X: Start signal
s_stConfig.stDoMachineX_Start.bCfgInvert := FALSE;
s_fbDoMachineX_Start(
	//i_bReqOutput	:= , // Set at sequencers 
	i_rstConfig	:= s_stConfig.stDoMachineX_Start);

// Machine X: Speed signal
s_fbAoMachineX_Speed(
	//i_fValue	:= ,// Set at sequencers 
	i_rstConfig	:= s_stConfig.stAoMachineX_Speed);
	
// Red light	
s_fbRedLight(
	i_bReqLightOn		:= s_bStaStateOfSomething,
	i_bReqFlashLight	:= s_bStaStateOfSomething2,
	i_rstConfig			:= s_stConfig.stRedLight);
END_METHOD

METHOD PROTECTED _m_Starting
VAR_INPUT
	i_rstPML_Status			: REFERENCE TO ST_PackML_Status;
END_VAR
VAR_INST
	s_fbSeqControl				: FB_SeqControl;
	s_eSeqAutoStarting			: E_EM_LogicExample1_Seq_StartingProduction;
	s_eActMode					: E_PackML_Mode;
END_VAR
// Execute only when in a specific mode
s_eActMode := i_rstPML_Status.eActMode;
IF i_rstPML_Status.eActMode = E_PackML_Mode.Production OR i_rstPML_Status.eActMode = E_PackML_Mode.UserMode1 THEN

	s_fbSeqControl(
		i_bReqStart		:= i_rstPML_Status.bStateEntry, 
		i_rnActSeqStep	:= s_eSeqAutoStarting,
		i_sActSeqStep	:= TO_STRING(s_eSeqAutoStarting));
	
		
	CASE s_eSeqAutoStarting OF
		E_EM_LogicExample1_Seq_StartingProduction.Idle:
			;
	
			
		E_EM_LogicExample1_Seq_StartingProduction.Start:	
			//Enable both axes in one singe sequencer step
			IF s_cmVirtualMaster.m_Enable() 
				AND s_cmAxis1.m_Enable()
			THEN
				s_fbSeqControl.m_ReqStep(E_EM_LogicExample1_Seq_StartingProduction.ReferenceAxes);
			END_IF
			
			
		E_EM_LogicExample1_Seq_StartingProduction.ReferenceAxes:	
			//Reference when needed both axes in one singe sequencer step
			//Both methode give a TRUE when the axis is referenced
			//i_bForceReference := TRUE => The reference routine is allways started even when the axis is allready referenced
			//i_bForceReference := FALSE => The refference routine is only started when the axis is not already referenced
			//Recommended is to reference virtual axis allways and real axis only when they has loses the reference state		
			IF s_cmVirtualMaster.m_ReferenceDrive(i_bCmdReset:= s_fbSeqControl.q_bStaEntry, i_bForceReference:=TRUE)
				AND s_cmAxis1.m_ReferenceDrive(i_bCmdReset:= s_fbSeqControl.q_bStaEntry, i_bForceReference:=FALSE)
			THEN
				// No camming License to store a cam-table
				//s_fbSeqControl.m_ReqStep(E_EM_LogicExample1_Seq_AutoStarting.CamAxis);
				s_fbSeqControl.m_ReqStep(E_EM_LogicExample1_Seq_StartingProduction.Ready);
			END_IF
		
			
		E_EM_LogicExample1_Seq_StartingProduction.CamAxis:
			//Cam in the slave (real axis) to the master axis
			//The Cam function is a methode of the camming Addon.
			//The methode give a TRUE when the Cam In is done.
			IF s_cmAxis1Cam.m_CamIn(
					i_bCmdReset					:= s_fbSeqControl.q_bStaEntry,
					i_fMasterOffset				:= 0.0,
					i_fSlaveOffset				:= 0.0,
					i_fMasterScale				:= 1,
					i_fSlaveScale				:= 1,
					i_bMasterOffsetIsRelative	:= FALSE,
					i_bSlaveOffsetIsRelative	:= FALSE,
					i_nCamTableId				:= nCamTableIdAxis1, 
					i_fMasterActivationPos		:= 0, 
					i_mcCamOperationMode		:= MC_CamOperationMode.CAMOPERATIONMODE_EXCHANGE,
					i_nReferenceCamTableID		:= 0,
					i_mcCamActivationMode		:= MC_CamActivationMode.MC_CAMACTIVATION_INSTANTANEOUS,
					i_mcMasterScalingMode		:= MC_CamScalingMode.MC_CAMSCALING_USERDEFINED,
					i_mcSlaveScalingMode		:= MC_CamScalingMode.MC_CAMSCALING_USERDEFINED,
					i_itfMaster					:= s_cmVirtualMaster)
			THEN
				s_fbSeqControl.m_ReqStep(E_EM_LogicExample1_Seq_StartingProduction.Ready);
			END_IF
			
			
		E_EM_LogicExample1_Seq_StartingProduction.Ready:
			;
			
			
		E_EM_LogicExample1_Seq_StartingProduction.Error:
			;
	
	END_CASE
		
	F_SeqControl_PackMLcommands(
		i_rnActSeqStep	:= s_eSeqAutoStarting,
		q_bStaFinished	=> i_rstPML_Status.bStateComplete,
		q_bStaIdle		=> ,
		q_bStaError		=> i_rstPML_Status.bStateError);
ELSE
	i_rstPML_Status.bStateComplete := TRUE;
END_IF
END_METHOD


METHOD PROTECTED _m_Starting_SubStates
VAR_INPUT
	i_rstPML_Status			: REFERENCE TO ST_PackML_Status;
END_VAR
VAR_INST
	s_fbSeqControl			: FB_SeqControl;
	s_eSeqAutoStarting		: E_EM_LogicExample1_Seq_StartingProduction;
	
	s_bStaDoneThis			: BOOL;
	s_bStaStateComplete1		: BOOL;
	s_bStaStateComplete2		: BOOL;
	s_bStaStateComplete3		: BOOL;
END_VAR
// Execute only when in a specific mode
CASE i_rstPML_Status.eActMode OF
	// Execute only when in PRODUCTION mode		
	E_PackML_Mode.Production: 
		CASE i_rstPML_Status.nActSubState OF
			1:
				s_bStaDoneThis := FALSE;
				i_rstPML_Status.bStateComplete := s_bStaStateComplete1;
			2:
				s_bStaDoneThis := TRUE;
				i_rstPML_Status.bStateComplete := s_bStaStateComplete2;
		ELSE
			i_rstPML_Status.bStateComplete := s_bStaStateComplete3;	
		END_CASE
		
	// Execute only when in MANUAL mode	
	E_PackML_Mode.Manual:
		i_rstPML_Status.bStateComplete := TRUE;
ELSE
	// Execute in all other modes	
	i_rstPML_Status.bStateComplete := TRUE;
END_CASE
END_METHOD

METHOD PROTECTED _m_Statistics
SUPER^._m_Statistics();

// Do all statistics here... Like fault counters or...

// Running times
// Belt
s_fbRunTime_Belt(
	i_bCmdReset		:= FALSE,
	i_bStaRunning	:= NOT s_cmBelt.q_bStaStandstill);
END_METHOD

METHOD PROTECTED _m_Stopping
VAR_INPUT
	i_rstPML_Status			: REFERENCE TO ST_PackML_Status;
END_VAR
VAR_INST
	
	s_bStaStateComplete1		: BOOL;
END_VAR
i_rstPML_Status.bStateComplete := _m_StopServos(i_bReqStart := i_rstPML_Status.bStateEntry);
END_METHOD

METHOD PRIVATE _m_StopServos : BOOL
VAR_INPUT
	i_bReqStart				: BOOL;			// Reset sequencer
END_VAR
VAR_INST
	s_fbSeqControl			: FB_SeqControl;
	s_eSeqCtrl_StopServos	: E_EM_LogicExample1_Seq_StopServos;
END_VAR
s_fbSeqControl(
	i_bReqStart		:= i_bReqStart, 
	i_rnActSeqStep	:= s_eSeqCtrl_StopServos,
	i_sActSeqStep	:= TO_STRING(s_eSeqCtrl_StopServos));

	
CASE s_eSeqCtrl_StopServos OF
	
	E_EM_LogicExample1_Seq_StopServos.Idle:
		;
		
	E_EM_LogicExample1_Seq_StopServos.Start:
		IF s_cmVirtualMaster.m_Stop(
			i_bCmdReset			:= s_fbSeqControl.q_bStaEntry,
			i_fDeceleration		:= s_cmVirtualMaster.q_stParameterSet.fDecelerationMax,
			i_fJerk				:= s_cmVirtualMaster.q_stParameterSet.fJerk) 
		AND
			s_cmAxis1.m_Stop(
				i_bCmdReset			:= s_fbSeqControl.q_bStaEntry,
				i_fDeceleration		:= s_cmAxis1.q_stParameterSet.fDecelerationMax,
				i_fJerk				:= s_cmAxis1.q_stParameterSet.fJerk) 
		THEN
			s_fbSeqControl.m_ReqStep(E_EM_LogicExample1_Seq_StopServos.Busy);
		END_IF
		
		//Add a time-out to be sure axis is disabled on time
		IF s_fbSeqControl.q_tmStepTime > T#100MS THEN
			s_fbSeqControl.m_ReqStep(E_EM_LogicExample1_Seq_StopServos.Busy);
		END_IF
		
	E_EM_LogicExample1_Seq_StopServos.Busy:	
		//Wait till axis is stopped. A time-out is added to sure that the axis is always disabled in on time		
		IF (s_cmVirtualMaster.q_stAxisState.StandStill 
			AND s_cmAxis1.q_stAxisState.StandStill) 
			OR s_fbSeqControl.q_tmStepTime > T#500MS 
		THEN
			s_cmVirtualMaster.m_Disable();
			s_cmAxis1.m_Disable();
			s_fbSeqControl.m_ReqStep(E_EM_LogicExample1_Seq_StopServos.Ready);
		END_IF
	
	E_EM_LogicExample1_Seq_StopServos.Ready:
		;

	E_EM_LogicExample1_Seq_StopServos.Error:
		;	

END_CASE


F_SeqControl_PackMLcommands(
	i_rnActSeqStep	:= s_eSeqCtrl_StopServos,
	q_bStaFinished	=> _m_StopServos,
	q_bStaIdle		=> ,
	q_bStaError		=> );
END_METHOD

{attribute 'monitoring' := 'call'}
PROPERTY p_bStaMachineX_Start_Active : BOOL
GET
p_bStaMachineX_Start_Active := s_fbDoMachineX_Start.q_bStaOutput;
END_GET
END_PROPERTY

{attribute 'monitoring' := 'call'}
PROPERTY p_bStaSensorPos1 : BOOL
GET
p_bStaSensorPos1 := s_fbDiSensorPos1.q_bStaInput;
END_GET
END_PROPERTY

{attribute 'monitoring' := 'call'}
PROPERTY p_itfCmAxis1 : ITF_CM_ServoBase
GET
p_itfCmAxis1 := s_cmAxis1;
END_GET
END_PROPERTY

{attribute 'monitoring' := 'call'}
PROPERTY p_itfCmBelt : ITF_CM_MotorDol
GET
p_itfCmBelt := s_cmBelt;
END_GET
END_PROPERTY

{attribute 'monitoring' := 'call'}
PROPERTY p_itfCmHeightAdjuster : ITF_CM_MotorDol_AF
GET
p_itfCmHeightAdjuster := s_cmHeightAdjuster;
END_GET
END_PROPERTY

{attribute 'monitoring' := 'call'}
PROPERTY p_itfCmWaterInlet : ITF_CM_Valve
GET
p_itfCmWaterInlet := s_cmWaterInlet;
END_GET
END_PROPERTY

{attribute 'monitoring' := 'call'}
PROPERTY p_rstConfig : REFERENCE TO ST_EM_LogicExample1_Config
GET
p_rstConfig := s_stConfig;
END_GET
END_PROPERTY

END_FUNCTION_BLOCK

(* stored: Version 1.1.0.1, ProductVersion 3.1.4024.10
   POU EM_LogicExample_1: Id {6f2f2bf2-c2da-4416-808c-ed5c6d63cc10}, SpecialFunc None
   Folder Basic: Id {4ed3fdc5-bc4f-4446-a28c-bed3cb0c11b8}
   Folder itfEM_LogicExample1: Id {0d3fe253-04f5-40ec-ac04-1fbfc387130a}
   Folder OMAC PackML: Id {b67bcd5d-8aa8-4ebc-a6e9-981237758fe2}
   Method _m_Aborting: Id {42785298-80cd-4aca-b777-b43d3b6adeba}
   Method _m_Alarms: Id {7e41031d-5a41-43de-945e-f69ca97b38b9}
   Method _m_Execute: Id {0a227c5f-6a54-4d0d-bf27-a184f6b93e6f}
   Method _m_Execute_Production: Id {e20eb719-ea1e-47b9-8aa3-fa6245349af8}
   Method _m_Init: Id {a109f297-b36b-4668-b63d-735900e0aeb6}
   Method _m_Inputs: Id {77e4728c-ffad-4128-a279-41c2d7615831}
   Method _m_Logic: Id {92a339b3-29f4-4403-8127-08fe7b3359cf}
   Method _m_Modules: Id {69768295-7443-40c1-8644-57ec9b3eff02}
   Method _m_Outputs: Id {46e775c6-9c73-43e1-b271-d1bbfcfc1dff}
   Method _m_Starting: Id {74bc4b2f-043a-4038-b439-df9753c56557}
   Method _m_Starting_SubStates: Id {400f85a2-e7d2-4436-aa22-f0a326fd6012}
   Method _m_Statistics: Id {46f84ba8-ec28-4c72-9159-35409bbaf08f}
   Method _m_Stopping: Id {f87d548b-0cad-4916-8130-e1f7b762eb18}
   Method _m_StopServos: Id {5b343d6e-2672-4004-945d-26825f09df86}
   Property p_bStaMachineX_Start_Active: Id {133ca14e-251f-40ef-b5a0-a1c8e9b6c38b}
   Get Get: Id {65cc60d6-5bff-4829-8e30-d4c564ca0f54}
   Property p_bStaSensorPos1: Id {5e3221d5-a26c-41db-9d99-610f1e5d3adc}
   Get Get: Id {0f779ed3-b327-419e-8ba5-ce3548eeb203}
   Property p_itfCmAxis1: Id {4b75f813-c9e5-4630-b9af-0d70f6f1bd52}
   Get Get: Id {90e3bac3-f3cf-4fa2-9327-08fa3ec9473d}
   Property p_itfCmBelt: Id {443e4b9a-33ef-4c12-a014-d7532db96e52}
   Get Get: Id {1231dc3f-7eb7-45bf-9bc9-88d647698073}
   Property p_itfCmHeightAdjuster: Id {c634e908-04ba-406e-9bc5-f977da81e4eb}
   Get Get: Id {a17d42a9-9ccd-456b-8159-4cd0a81d514e}
   Property p_itfCmWaterInlet: Id {09035550-cd1c-43a8-8c21-a59ee1f9efd0}
   Get Get: Id {9e072766-9ff5-44a2-98a7-6e04b7999869}
   Property p_rstConfig: Id {32e99255-cfbc-4c85-bd78-849b1d6713ae}
   Get Get: Id {0732c555-1ae1-4488-bcb4-99e18728ae24} *)
